(* PLC project Unnamed, Unknown Unnamed 1 *)
(* stored: creationDateTime 2026-04-23T14:19:54, modificationDateTime 2026-04-23T14:19:54 *)

FUNCTION_BLOCK OSC
  VAR_INPUT
    t : TIME;
  END_VAR
  VAR_OUTPUT
    out : BOOL;
  END_VAR
  VAR
    a : BOOL;
    TON0 : TON;
    TOF0 : TOF;
  END_VAR

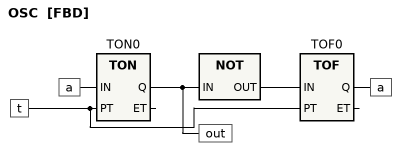
(* FBD diagram, written out as Structured Text *)
TON0(IN := a, PT := t);
out := TON0.Q;
TOF0(IN := NOT TON0.Q, PT := t);
a := TOF0.Q;
END_FUNCTION_BLOCK

PROGRAM main
  VAR
    Aumenta AT %QX0.0 : BOOL;
    Diminui AT %QX0.1 : BOOL;
    Contagem AT %QW0 : INT;
  END_VAR
  VAR
    OSC0 : OSC;
    CTUD0 : CTUD;
  END_VAR

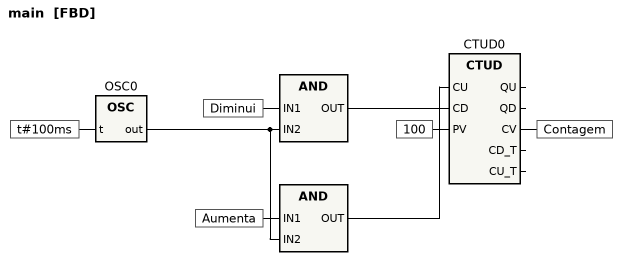
(* FBD diagram, written out as Structured Text *)
OSC0(t := t#100ms);
CTUD0(CU := Aumenta AND OSC0.out, CD := Diminui AND OSC0.out, PV := 100);
Contagem := CTUD0.CV;
END_PROGRAM

CONFIGURATION Config0
  RESOURCE Res0 ON PLC
    TASK task0(INTERVAL := T#20ms, PRIORITY := 1);
    PROGRAM instance0 WITH task0 : main;
  END_RESOURCE
END_CONFIGURATION
